INTERFACE I_ComponentVisitor

METHOD VisitComponent
VAR_INPUT
	Component : I_Component;
END_VAR
END_METHOD

END_INTERFACE

(* stored: Version 1.1.0.1, ProductVersion 3.1.4026.18
   Itf I_ComponentVisitor: Id {4447d1fa-8e11-4539-9271-466db2f8a98b}
   Method VisitComponent: Id {a4dca2db-a1da-40f4-be4c-71660239c2ab} *)
